FUNCTION_BLOCK E_MERGE_2 (* Merge (OR) of two input events (generic FB) *)
  {SET_ATTRIBUTE(eclipse4diac::core::GenericClassName, 'GEN_E_MERGE')}
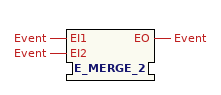
  EVENT_INPUT
    EI1; (* First input event *)
    EI2; (* Second input event *)
  END_EVENT
  EVENT_OUTPUT
    EO; (* Output Event *)
  END_EVENT
END_FUNCTION_BLOCK
